// TIA Portal project "Teste_Marcus" (V18)

(* hardware
DEVICE "S7-1200 station_1"  S7-1200 Station
   slot 0: "Rack_0"  S7-1200 Rack  Rack  V1.0
   slot 1: "PLC_1"  CPU 1214C AC/DC/Rly  6ES7 214-1BG40-0XB0  V4.5
   slot 2: "DI 16/DQ 16x24VDC_1"  6ES7 223-1BL32-0XB0  V2.0
   slot 3: "AI 8x13BIT_1"  6ES7 231-4HF32-0XB0  V2.1
*)

// ===== PLC "PLC_1"  CPU 1214C AC/DC/Rly =====

VAR_GLOBAL   // PLC tag table "Default tag table"
   "Tag_1" AT %Q0.6 : Bool;
   "Tag_2" AT %Q0.7 : Bool;
   "LED_Verde" AT %Q0.1 : Bool;
   "CH3" AT %I0.6 : Bool;
   "CH4" AT %I0.7 : Bool;
   "BL" AT %I0.1 : Bool;
   "LED_Vermelho" AT %Q0.3 : Bool;
   "LED_Amarelo" AT %Q0.0 : Bool;
   "BD" AT %I0.3 : Bool;
END_VAR

ORGANIZATION_BLOCK "Main"   // OB1, LAD, ProgramCycle
TITLE = "Main Program Sweep (Cycle)"
{ S7_Optimized_Access := 'TRUE' }
VERSION : 0.1
   VAR_INPUT
      Initial_Call : Bool;   // Initial call of this OB
      Remanence : Bool;   // =True, if remanent data are available
   END_VAR
BEGIN

REGION Network 1
   // Ações da Chave Seletora (CS)
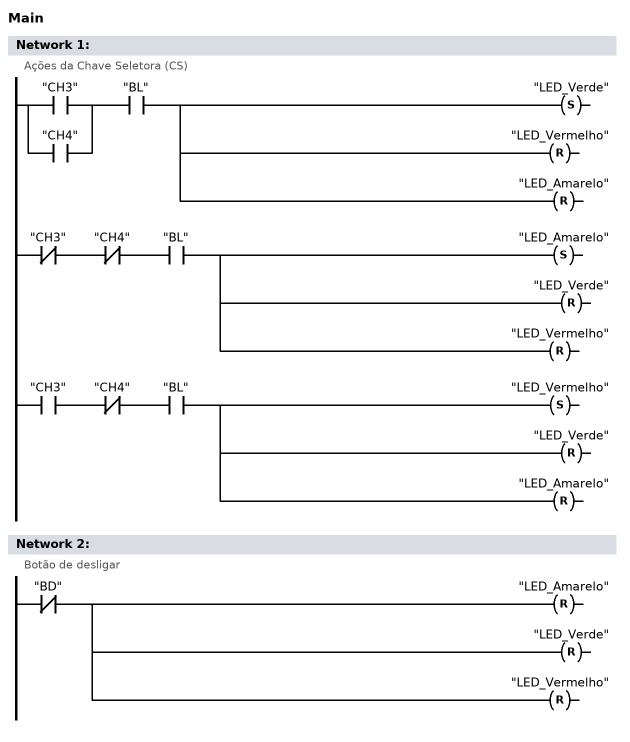
   RUNG wire#powerrail
      Contact( "CH3" )
      wire#w1
      Contact( "BL" )
      wire#w2
      S_Coil( "LED_Verde" )
   END_RUNG
   RUNG wire#powerrail
      Contact( "CH4" )
   END_RUNG wire#w1
   RUNG wire#w2
      R_Coil( "LED_Vermelho" )
   END_RUNG
   RUNG wire#w2
      R_Coil( "LED_Amarelo" )
   END_RUNG
   RUNG wire#powerrail
      I_Contact( "CH3" )
      I_Contact( "CH4" )
      Contact( "BL" )
      wire#w3
      S_Coil( "LED_Amarelo" )
   END_RUNG
   RUNG wire#w3
      R_Coil( "LED_Verde" )
   END_RUNG
   RUNG wire#w3
      R_Coil( "LED_Vermelho" )
   END_RUNG
   RUNG wire#powerrail
      Contact( "CH3" )
      I_Contact( "CH4" )
      Contact( "BL" )
      wire#w4
      S_Coil( "LED_Vermelho" )
   END_RUNG
   RUNG wire#w4
      R_Coil( "LED_Verde" )
   END_RUNG
   RUNG wire#w4
      R_Coil( "LED_Amarelo" )
   END_RUNG
   // the same network as SCL:
   IF ("CH3" OR "CH4") AND "BL" THEN
       "LED_Verde" := TRUE;
       "LED_Vermelho" := FALSE;
       "LED_Amarelo" := FALSE;
   END_IF;
   IF NOT "CH3" AND NOT "CH4" AND "BL" THEN
       "LED_Amarelo" := TRUE;
       "LED_Verde" := FALSE;
       "LED_Vermelho" := FALSE;
   END_IF;
   IF "CH3" AND NOT "CH4" AND "BL" THEN
       "LED_Vermelho" := TRUE;
       "LED_Verde" := FALSE;
       "LED_Amarelo" := FALSE;
   END_IF;
END_REGION

REGION Network 2
   // Botão de desligar
   RUNG wire#powerrail
      I_Contact( "BD" )
      wire#w1
      R_Coil( "LED_Amarelo" )
   END_RUNG
   RUNG wire#w1
      R_Coil( "LED_Verde" )
   END_RUNG
   RUNG wire#w1
      R_Coil( "LED_Vermelho" )
   END_RUNG
   // the same network as SCL:
   IF NOT "BD" THEN
       "LED_Amarelo" := FALSE;
       "LED_Verde" := FALSE;
       "LED_Vermelho" := FALSE;
   END_IF;
END_REGION
END_ORGANIZATION_BLOCK